// function block for reed switch with the option of debouncing + rising and falling edge detection.
FUNCTION_BLOCK FB_ReedSwitch IMPLEMENTS I_Component
VAR_INPUT
	bSignal			: BOOL;				// Raw input sensor
	tDebounce		: TIME := T#0MS;	// Debounce time
// Interface vars
	sName			: STRING[20];
	bEnable     	: BOOL;
	//eMode       	: E_ComponentMode;
END_VAR

VAR_OUTPUT
	bActive			: BOOL;
	bRising			: BOOL;
	bFalling		: BOOL;
// interface vars
	eState			: E_ComponentState;
	iErrorCode		: INT;
	sStatusText 	: STRING[50];
END_VAR

VAR
	bLastSignal		: BOOL;
	tDebTimer		: TON;
	bSignalStable	: BOOL;
END_VAR

IF bEnable AND eState = (E_ComponentState.READY OR E_ComponentState.BUSY) THEN
	IF bLastSignal <> bSignal THEN
		tDebTimer(IN := TRUE, PT := tDebounce);
		eState := E_ComponentState.BUSY;
	ELSE
		tDebTimer(IN := FALSE);
	END_IF
	
	IF tDebTimer.Q THEN
		bSignalStable 	:= bSignal;
		bLastSignal 	:= bSignal;
		eState := E_ComponentState.READY;
	END_IF
	
	bRising		:= (bSignalStable AND NOT bActive);
	bFalling	:= (NOT bSignalStable AND bActive);
	bActive 	:= bSignalStable;
ELSE
	bActive 	:= FALSE;
	bRising		:= FALSE;
	bFalling	:= FALSE;
	tDebTimer(IN := FALSE);
END_IF

METHOD Halt : BOOL
VAR_INPUT
END_VAR
bActive 	:= FALSE;
bRising		:= FALSE;
bFalling	:= FALSE;
tDebTimer(IN := FALSE);
eState := E_ComponentState.HALTED;
END_METHOD

METHOD Start : BOOL
VAR_INPUT
END_VAR
eState := E_ComponentState.READY;
END_METHOD

METHOD Stop : BOOL
VAR_INPUT
END_VAR
IF eState <> E_ComponentState.BUSY THEN
	bActive 	:= FALSE;
	bRising		:= FALSE;
	bFalling	:= FALSE;
	eState := E_ComponentState.DONE;
END_IF
END_METHOD

END_FUNCTION_BLOCK

(* stored: Version 1.1.0.1, ProductVersion 3.1.4024.15
   POU FB_ReedSwitch: Id {f639b4a8-9d3e-46fd-a4ee-568d4dd5739a}, SpecialFunc None
   Method Halt: Id {c94396e9-4b2a-428e-b504-c709afbc748b}
   Method Start: Id {3ee6110b-c203-4bb9-9caa-b0b18392f854}
   Method Stop: Id {60cdd494-a322-4122-a75f-cf6898b5dc26} *)
